// TIA Portal V18 export
DATA_BLOCK "FC1520_EZO_TCPClient_DB"   // DB6
VERSION : 0.1
// stored: AutoNumber true, DBAccessibleFromOPCUA true, DBAccessibleFromWebserver true, InstanceOfName FB1520_EZO_TCPClient, InstanceOfType FB
"FB1520_EZO_TCPClient"
   // VAR_INPUT
   //    Enable : Bool;
   //    EN_R : Bool;
   //    ID : CONN_OUC;
   //    PORT : UInt;
   //    IP_1 : Byte;
   //    IP_2 : Byte;
   //    IP_3 : Byte;
   //    IP_4 : Byte;
   // END_VAR
   // VAR_OUTPUT
   //    DONE : Bool;
   //    BUSY : Bool;
   //    ERROR : Bool;
   //    STATUS : Word;
   //    Value : Real;
   // END_VAR
   // VAR_IN_OUT
   //    COM_RST : Bool;
   // END_VAR
   // VAR
   //    CONNECT : TCON_IP_v4;
   //    RCV_DATA : Array[0..8] of Char;
   //    Done_Old : Bool;
   //    Pos_R : Int;
   //    TRCV_C1 : TRCV_C;
   //    QT1 { S7_SetPoint := 'True'} : Bool;
   //    QT2 : Bool;
   //    T1 { S7_SetPoint := 'True'} : TON_TIME;
   //    T2 { S7_SetPoint := 'True'} : TON_TIME;
   // END_VAR
BEGIN
END_DATA_BLOCK
